{attribute 'linkalways'} 
{attribute 'no_explicit_call' := 'This FB is a CLASS and must be accessed using methods or properties'}
{attribute 'enable_dynamic_creation'}
FUNCTION_BLOCK FINAL EXP_LREAL EXTENDS Node
VAR
	in : _LREAL(0.0);
	out : _LREAL(0.0);
END_VAR

METHOD PUBLIC Clone : I_Node
VAR
	pNode : POINTER TO EXP_LREAL;
END_VAR
pNode := __NEW(EXP_LREAL);
Clone := pNode^;
END_METHOD

METHOD FB_init : BOOL
VAR_INPUT
	bInitRetains : BOOL; // if TRUE, the retain variables are initialized (warm start / cold start)
	bInCopyCode : BOOL;  // if TRUE, the instance afterwards gets moved into the copy code (online change)
END_VAR
AddInput('in',THIS^.in);
AddOutput('out', THIS^.out);
END_METHOD

METHOD PROTECTED OnExecute
VAR
END_VAR
out.Value := EXP(in.Value);
END_METHOD

END_FUNCTION_BLOCK

(* stored: Version 1.1.0.1, ProductVersion 3.1.4024.15
   POU EXP_LREAL: Id {4e43f1be-f7f0-49e2-96c1-ca9eafdaca42}, SpecialFunc None
   Folder Constructor: Id {14c87cd5-bf78-4831-a8d0-0a60ea3a7290}
   Method Clone: Id {c83cd457-01d4-4ba8-88db-e4d34b3a0bda}
   Method FB_init: Id {b7570be8-375c-4e3a-ae42-d0fca1ca9312}
   Method OnExecute: Id {5128ce39-b961-427e-baa2-7cbe750c7655} *)
